SUBAPPLICATION Uebung_086 (* Beispiel für E_SWITCH *)
  (* Standard: 61499-2; Description: Copyright (c) 2023 Meisterschulen am Ostbahnhof This program and the accompanying materials are made available under the terms of the Eclipse Public License 2.0 which is available at https://www.eclipse.org/legal/epl-2.0/ SPDX-License-Identifier: EPL-2.0 Beispiel für E_CTD Aufwärts zählen UAO Curriculum Module 3 - The IEC 61499 Standard, Seite 93 *)
  (* Version 1.0, 2023-10-23, Franz Höpfinger, Meisterschulen am Ostbahnhof *)
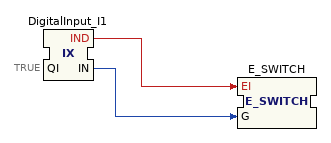
  FBS
    DigitalInput_I1 : IX(QI := TRUE);
    E_SWITCH : E_SWITCH;
  END_FBS
  EVENT_CONNECTIONS
    DigitalInput_I1.IND TO E_SWITCH.EI;
  END_CONNECTIONS
  DATA_CONNECTIONS
    DigitalInput_I1.IN TO E_SWITCH.G;
  END_CONNECTIONS
END_SUBAPPLICATION
